FUNCTION_BLOCK FB_PU_191_Ablaufsteuerung
VAR_IN_OUT
	Zustand			: ST_PU_Zustand;
	Stellwert			: ST_PU_Stellwert;
END_VAR
VAR_INPUT
	Steuerung		: ST_PU_Steuerung;
	Parameter		: ST_PU_Parameter;
END_VAR
VAR_OUTPUT
END_VAR
VAR
	Timer			: TON;
END_VAR

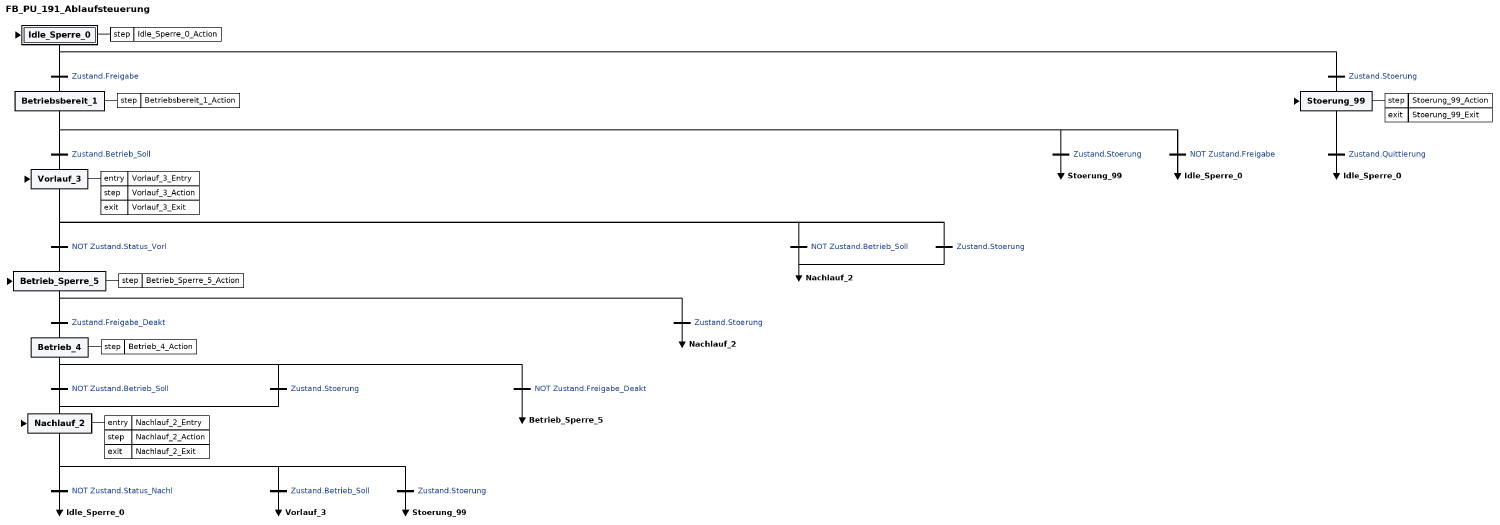
INITIAL_STEP Idle_Sperre_0:
    Idle_Sperre_0_Action(N);  // step action
END_STEP
TRANSITION FROM Idle_Sperre_0 TO Betriebsbereit_1
    := Zustand.Freigabe;
END_TRANSITION
TRANSITION FROM Idle_Sperre_0 TO Stoerung_99
    := Zustand.Stoerung;
END_TRANSITION
STEP Stoerung_99:
    Stoerung_99_Action(N);  // step action
    Stoerung_99_Exit(P0);  // exit action
END_STEP
TRANSITION FROM Stoerung_99 TO Idle_Sperre_0
    := Zustand.Quittierung;
END_TRANSITION
STEP Betriebsbereit_1:
    Betriebsbereit_1_Action(N);  // step action
END_STEP
TRANSITION FROM Betriebsbereit_1 TO Vorlauf_3
    := Zustand.Betrieb_Soll;
END_TRANSITION
TRANSITION FROM Betriebsbereit_1 TO Stoerung_99
    := Zustand.Stoerung;
END_TRANSITION
TRANSITION FROM Betriebsbereit_1 TO Idle_Sperre_0
    := NOT Zustand.Freigabe;
END_TRANSITION
STEP Vorlauf_3:
    Vorlauf_3_Entry(P1);  // entry action
    Vorlauf_3_Action(N);  // step action
    Vorlauf_3_Exit(P0);  // exit action
END_STEP
TRANSITION FROM Vorlauf_3 TO Betrieb_Sperre_5
    := NOT Zustand.Status_Vorl;
END_TRANSITION
TRANSITION FROM Vorlauf_3 TO Nachlauf_2
    := NOT Zustand.Betrieb_Soll;
END_TRANSITION
TRANSITION FROM Vorlauf_3 TO Nachlauf_2
    := Zustand.Stoerung;
END_TRANSITION
STEP Betrieb_Sperre_5:
    Betrieb_Sperre_5_Action(N);  // step action
END_STEP
TRANSITION FROM Betrieb_Sperre_5 TO Betrieb_4
    := Zustand.Freigabe_Deakt;
END_TRANSITION
TRANSITION FROM Betrieb_Sperre_5 TO Nachlauf_2
    := Zustand.Stoerung;
END_TRANSITION
STEP Betrieb_4:
    Betrieb_4_Action(N);  // step action
END_STEP
TRANSITION FROM Betrieb_4 TO Nachlauf_2
    := NOT Zustand.Betrieb_Soll;
END_TRANSITION
TRANSITION FROM Betrieb_4 TO Nachlauf_2
    := Zustand.Stoerung;
END_TRANSITION
TRANSITION FROM Betrieb_4 TO Betrieb_Sperre_5
    := NOT Zustand.Freigabe_Deakt;
END_TRANSITION
STEP Nachlauf_2:
    Nachlauf_2_Entry(P1);  // entry action
    Nachlauf_2_Action(N);  // step action
    Nachlauf_2_Exit(P0);  // exit action
END_STEP
TRANSITION FROM Nachlauf_2 TO Idle_Sperre_0
    := NOT Zustand.Status_Nachl;
END_TRANSITION
TRANSITION FROM Nachlauf_2 TO Vorlauf_3
    := Zustand.Betrieb_Soll;
END_TRANSITION
TRANSITION FROM Nachlauf_2 TO Stoerung_99
    := Zustand.Stoerung;
END_TRANSITION

ACTION Betrieb_4_Action:
(* Stellwert setzen *)
Stellwert.Betrieb := TRUE;

(* Zustand setzen *)
Zustand.Status := E_PU_Zustand_Status_Betrieb;
END_ACTION

ACTION Betrieb_Sperre_5_Action:
(* Stellwert setzen *)
Stellwert.Betrieb := TRUE;

(* Zustand setzen *)
Zustand.Status := E_PU_Zustand_Status_Betrieb_Sperre;
END_ACTION

ACTION Betriebsbereit_1_Action:
(* Stellwert setzen *)
Stellwert.Betrieb := FALSE;

(* Zustand setzen *)
Zustand.Status := E_PU_Zustand_Status_Betriebsbereit;
END_ACTION

ACTION Idle_Sperre_0_Action:
(* Stellwert setzen *)
Stellwert.Betrieb := FALSE;

(* Zustand setzen *)
Zustand.Status := E_PU_Zustand_Status_Idle_Sperre;
END_ACTION

ACTION Nachlauf_2_Action:
(* Nachlauf Timer starten *)
Timer( 	IN := Zustand.Status_Nachl,
		PT := DINT_TO_TIME(Parameter.Zeit_Nachl)
);
Zustand.Status_Nachl	:= NOT(Timer.Q AND NOT Zustand.Betrieb);

(* Stellwert setzen *)
Stellwert.Betrieb := FALSE;

(* Zustand setzen *)
Zustand.Status := E_PU_Zustand_Status_Nachl;
END_ACTION

ACTION Nachlauf_2_Entry:
(* Reset Timer *)
Timer(IN := FALSE);
Zustand.Status_Nachl := TRUE;
END_ACTION

ACTION Nachlauf_2_Exit:
Zustand.Status_Nachl := FALSE;
END_ACTION

ACTION Stoerung_99_Action:
(* Stellwert setzen *)
Stellwert.Betrieb := FALSE;

(* Zustand setzen *)
Zustand.Stoerung := TRUE;
Zustand.Status := E_PU_Zustand_Status_Stoerung;
END_ACTION

ACTION Stoerung_99_Exit:
Zustand.Stoerung	:= FALSE;
END_ACTION

ACTION Vorlauf_3_Action:
(* Vorlaufzeit Timer starten *)
Timer( 	IN := Zustand.Status_Vorl,
		PT := DINT_TO_TIME(Parameter.Zeit_Vorl)
);
Zustand.Status_Vorl := NOT (Timer.Q AND Zustand.Betrieb);

(* Stellwert setzen *)
Stellwert.Betrieb := TRUE;

(* Zustand setzen *)
Zustand.Status := E_PU_Zustand_Status_Vorl;
END_ACTION

ACTION Vorlauf_3_Entry:
(* Reset Timer *)
Timer(IN := FALSE);
Zustand.Status_Vorl := TRUE;
END_ACTION

ACTION Vorlauf_3_Exit:
Zustand.Status_Vorl := FALSE;
END_ACTION

END_FUNCTION_BLOCK

(* stored: Version 1.1.0.1, ProductVersion 3.1.4024.9
   POU FB_PU_191_Ablaufsteuerung: Id {3b35f71a-5af5-4f7b-b9e5-8f895ca2c237}, SpecialFunc None
   Action Betrieb_4_Action: Id {b1222823-5b66-43ba-88eb-1db09e5ce93e}
   Action Betrieb_Sperre_5_Action: Id {4e96cde1-ebd3-4155-92d4-163cefe71763}
   Action Betriebsbereit_1_Action: Id {c2851b12-77e3-44bf-9e77-2a2e0604ac67}
   Action Idle_Sperre_0_Action: Id {71193604-26e2-4610-a02b-b4a44de830b2}
   Action Nachlauf_2_Action: Id {547a31d0-ace2-41c0-bc4f-9a611f3742cc}
   Action Nachlauf_2_Entry: Id {392feaeb-dfff-4e50-9376-587452263031}
   Action Nachlauf_2_Exit: Id {8a811395-d371-4e88-b49c-d4386c8d23af}
   Action Stoerung_99_Action: Id {35d91b67-259f-44d9-80d8-e639d5d90ca7}
   Action Stoerung_99_Exit: Id {a0e3f9ed-4f64-406f-a792-86233ab07eb6}
   Action Vorlauf_3_Action: Id {3c10e6c9-d135-4614-b6fc-76b4dc6dd645}
   Action Vorlauf_3_Entry: Id {f5da5e04-cda2-4b14-aebb-a85859eee0e6}
   Action Vorlauf_3_Exit: Id {694c995a-88a8-4057-84a9-6dfc7e1268c3} *)
